// TIA Portal V19 export
VAR_GLOBAL   // PLC tag table "U3Em1_output"
   ngBeltBackLight AT %Q1.3 : Bool;
   ngBeltForwardLight AT %Q1.2 : Bool;
END_VAR
